FUNCTION_BLOCK GEN_SQR (* this signal generator generates a square wave output *)
  (* Standard: 61499-1; Description: version 1.4	11. mar. 2009 programmer 	oscat tested BY		oscat this signal generator generates a square wave output. The square wave signal is defined by period time (PT), amplitude (AM), offset (OS), duty cycle (DC) and a specific delay for the output signal (DL). The Output waveform will switch between AM/2 + OS and -AM/2 + OS. The DC input specifies ther duty cycle, DC = 0 means output is low at all times and 1 means output is high at all times. The delay input can delay a signal up to PT, this can be useful to synchronize different generators and generate interleaving signals. in addition to a analog output Out there is a second boolean output Q. *)
  (* Version 1.0, 2025-12-21, Franz Höpfinger, initial API and implementation and/or initial documentation *)
  PACKAGE OSCAT::Basic::POUs::Engineering::signal_generators;
  IMPORT OSCAT::Basic::POUs::Mathematical::MODR;
  IMPORT OSCAT::Basic::POUs::Time_Date::MULTIME;
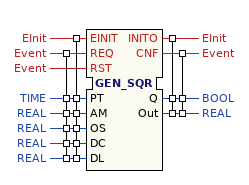
  EVENT_INPUT
    EINIT : EInit WITH PT, AM, OS, DC, DL; (* Init Request *)
    REQ WITH PT, AM, OS, DC, DL; (* Normal Execution Request *)
    RST; (* Reset *)
  END_EVENT
  EVENT_OUTPUT
    INITO : EInit WITH Q, Out; (* Init Confirmation *)
    CNF WITH Q, Out; (* Execution Confirmation *)
  END_EVENT
  VAR_INPUT
    PT : TIME; (* Period Time *)
    AM : REAL := 1.0; (* Amplitude *)
    OS : REAL; (* Offset *)
    DC : REAL := 0.5; (* Duty Cycle *)
    DL : REAL; (* Delay *)
  END_VAR
  VAR_OUTPUT
    Q : BOOL; (* Pulse Output *)
    Out : REAL; (* Signal Output *)
  END_VAR
  VAR
    tx : TIME;
    last : TIME;
    init : BOOL;
    DL_M : REAL;
    DC_M : REAL;
  END_VAR
  EC_STATES
    EINIT : EINIT -> INITO;
    REQ : REQ -> CNF;
    RST : RST -> CNF;
  END_STATES
  ALGORITHM EINIT IN ST:
init := FALSE;
  END_ALGORITHM
  ALGORITHM RST IN ST:
init := TRUE;
last := tx;
tx := T#0s;
  END_ALGORITHM
  ALGORITHM REQ IN ST:
(* check dc = 1 or 0 *)
IF DC = 0.0 THEN
	Out := -AM * 0.5 + OS;
	Q := FALSE;
	RETURN;
ELSIF DC = 1.0 THEN
	Out := AM * 0.5 + OS;
	Q := TRUE;
	RETURN;
END_IF;

(* read system time and prepare input data *)
tx := NOW_MONOTONIC() - last;
DL_M := MODR(DL, 1.0);
IF DL_M < 0.0 THEN
	DL_M := 1.0 - DL_M;
END_IF;
DC_M := MODR(DC, 1.0);
IF DC_M < 0.0 THEN
	DC_M := 1.0 - DC_M;
END_IF;

(* init section *)
IF NOT init THEN
	this.RST();
END_IF;

(* add last if one cycle is finished *)
IF tx >= PT THEN
	last := last + PT;
	tx := tx - PT;
END_IF;

(* check if falling or rising edge first *)
IF MULTIME(PT, DL + DC) >= PT THEN
	(* generate falling edge *)
	IF tx >= MULTIME(PT, DL + DC - 1.0) THEN
		Out := -AM * 0.5 + OS;
		Q := FALSE;
	END_IF;
	(* generate rising edge *)
	IF tx >= MULTIME(PT, DL) THEN
		Out := AM * 0.5 + OS;
		Q := TRUE;
	END_IF;
ELSE
	(* generate rising edge first *)
	IF tx >= MULTIME(PT, DL) THEN
		Out := AM * 0.5 + OS;
		Q := TRUE;
	END_IF;
		(* generate falling edge *)
	IF tx >= MULTIME(PT, DL + DC) THEN
		Out := -AM * 0.5 + OS;
		Q := FALSE;
	END_IF;
END_IF;
  END_ALGORITHM
END_FUNCTION_BLOCK
